{region '#Template'}
	{attribute 'Category' := 'General'}
	{attribute 'Version' := '0.0.1.0'}
	{attribute 'Tags' := 'General, Cabinet, Control cabinet'}
	{attribute 'Description' := 'Schaltschrank Ereignisse	// Control cabinet events'}
{endregion}
FUNCTION_BLOCK FB_BA_ControlCabinet EXTENDS FB_BA_ControlCabinetBasic
VAR_INPUT CONSTANT
	Fuse01					: FB_BA_SensorBinary_IO;		
	Fuse02					: FB_BA_SensorBinary_IO;	
	Fuse03					: FB_BA_SensorBinary_IO;	
END_VAR

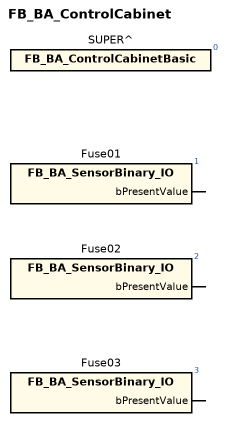
SUPER^(); // FB_BA_ControlCabinetBasic
Fuse01(); // FB_BA_SensorBinary_IO
Fuse02(); // FB_BA_SensorBinary_IO
Fuse03(); // FB_BA_SensorBinary_IO

METHOD FB_init : BOOL
VAR_INPUT
	bInitRetains : BOOL; // if TRUE, the retain variables are initialized (warm start / cold start)
	bInCopyCode : BOOL;  // if TRUE, the instance afterwards gets moved into the copy code (online change)
END_VAR
Fuse01.iParent								:= THIS^;		
Fuse01.iLabel 								:= LblCmpGeneral.ControlCabinet_Fuse;	
Fuse01.sObjectName							:= '{Idx=01}';
Fuse01.eDPADMode							:= E_BA_DPADMode.eInclude;																						
Fuse01.Input.iLabel							:= LblCmpGeneral.ControlCabinet_Fuse_Input;	
Fuse01.Input.sObjectName					:= '{Idx=01}';	
Fuse01.Input.ePolarity						:= E_BA_Polarity.eReverse;
Fuse01.Input.sActiveText 					:= Texts.txtTriggered;
Fuse01.Input.sInactiveText 					:= Texts.txtNormal;
Fuse01.Input.nEventClassID					:= EventClasses.AlarmTechnicalExtended;
Fuse01.Input.aEventTransitionText[1]		:= Texts.txtTriggered;
Fuse01.Input.aEventTransitionText[2]		:= Texts.txtError;
Fuse01.Input.aEventTransitionText[3]		:= Texts.txtNormal;
Fuse01.Input.bEventDetectionEnable			:= TRUE;
Fuse01.Input.eEnPlantLock					:= E_BA_LockPriority.eNoLock;	
								 
Fuse02.iParent								:= THIS^;		
Fuse02.iLabel 								:= LblCmpGeneral.ControlCabinet_Fuse;	
Fuse02.sObjectName							:= '{Idx=02}';
Fuse02.eDPADMode							:= E_BA_DPADMode.eInclude;																						
Fuse02.Input.iLabel							:= LblCmpGeneral.ControlCabinet_Fuse_Input;	
Fuse02.Input.sObjectName					:= '{Idx=02}';	
Fuse02.Input.ePolarity						:= E_BA_Polarity.eReverse;
Fuse02.Input.sActiveText 					:= Texts.txtTriggered;
Fuse02.Input.sInactiveText 					:= Texts.txtNormal;
Fuse02.Input.nEventClassID					:= EventClasses.AlarmTechnicalExtended;
Fuse02.Input.aEventTransitionText[1]		:= Texts.txtTriggered;
Fuse02.Input.aEventTransitionText[2]		:= Texts.txtError;
Fuse02.Input.aEventTransitionText[3]		:= Texts.txtNormal;
Fuse02.Input.bEventDetectionEnable			:= TRUE;
Fuse02.Input.eEnPlantLock					:= E_BA_LockPriority.eNoLock;	
										 
Fuse03.iParent								:= THIS^;		
Fuse03.iLabel 								:= LblCmpGeneral.ControlCabinet_Fuse;	
Fuse03.sObjectName							:= '{Idx=03}';
Fuse03.eDPADMode							:= E_BA_DPADMode.eInclude;																						
Fuse02.Input.iLabel							:= LblCmpGeneral.ControlCabinet_Fuse_Input;	
Fuse02.Input.sObjectName					:= '{Idx=03}';	
Fuse02.Input.ePolarity						:= E_BA_Polarity.eReverse;
Fuse02.Input.sActiveText 					:= Texts.txtTriggered;
Fuse02.Input.sInactiveText 					:= Texts.txtNormal;
Fuse02.Input.nEventClassID					:= EventClasses.AlarmTechnicalExtended;
Fuse02.Input.aEventTransitionText[1]		:= Texts.txtTriggered;
Fuse02.Input.aEventTransitionText[2]		:= Texts.txtError;
Fuse02.Input.aEventTransitionText[3]		:= Texts.txtNormal;
Fuse02.Input.bEventDetectionEnable			:= TRUE;
Fuse02.Input.eEnPlantLock					:= E_BA_LockPriority.eNoLock;
END_METHOD

END_FUNCTION_BLOCK

(* stored: Version 1.1.0.1, ProductVersion 3.1.4024.6
   POU FB_BA_ControlCabinet: Id {b472c277-a5c6-4cc3-9f14-f22f885bb717}, SpecialFunc None
   Method FB_init: Id {907425df-4e48-49e5-919a-3e08157b204c} *)
